Fanuc KAREL source: ka00185.KL

PROGRAM KA00185
%STACKSIZE=65535
%PRIORITY=65535
%NOLOCKGROUP
-- UNRESOLVED DECLARATIONS (source type spelling not recovered)
-- SRC : ARRAY[4] OF TYPE_0x0018 (type_u16=0x2018)
-- DST : ARRAY[4] OF TYPE_0x0018 (type_u16=0x2018)
BEGIN
-- UNRESOLVED_PC line 7 opcodes [22 22 1E] marker_code=0
END KA00185
